FUNCTION FC_ScaleValue : LREAL
VAR_INPUT
	rangeRawMin		: LREAL;
	rangeRawMax		: LREAL;
	ValueRaw		: LREAL;
	RangeScaleMin	: LREAL;
	RangeScaleMax	: LREAL;
 
END_VAR
VAR
END_VAR

IF (rangeRawMax-rangeRawMin) < 0.0000001 THEN
	FC_ScaleValue := 0;
ELSE
	FC_ScaleValue := ((ValueRaw-rangeRawMin)/(rangeRawMax-rangeRawMin)) *(RangeScaleMax-RangeScaleMin) + RangeScaleMin;
END_IF

END_FUNCTION

(* stored: Version 1.1.0.1, ProductVersion 3.1.4024.12
   POU FC_ScaleValue: Id {a937f20d-2f08-4f64-8a08-e36bedbb68bd}, SpecialFunc None *)
